Xinje XDPPro project, PLC1: XD3-48 (software 3.8.0 2025-09-09)

PROGRAM Ladder

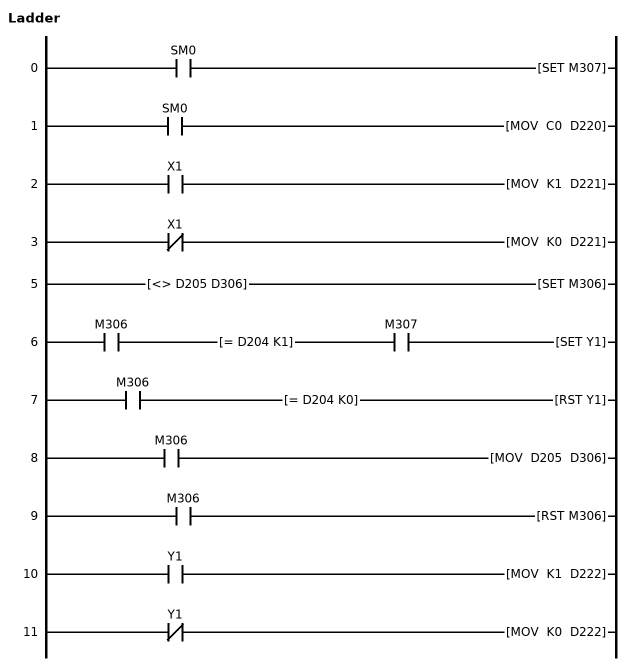
LD     SM0
SET    M307
LD     SM0
MOV    C0 D220
LD     X1
MOV    K1 D221
LDI    X1
MOV    K0 D221
LD<>   D205 D306
SET    M306
LD     M306
AND=   D204 K1
AND    M307
SET    Y1
LD     M306
AND=   D204 K0
RST    Y1
LD     M306
MOV    D205 D306
LD     M306
RST    M306
LD     Y1
MOV    K1 D222
LDI    Y1
MOV    K0 D222